FUNCTION TFWAconCodiceWPPPresente : BOOL // Valuta se esiste una WA in lavorazione con il codice del pacco sul ribaltino, se esiste ritorna true, altrimenti false
VAR_INPUT
	WorkArea : POINTER TO ARRAY [1..MAXAREA] OF TFMachinePalletizer_WorkArea;
	WorkAreaState : POINTER TO ARRAY [1..MAXAREA] OF TFMachinePalletizer_WorkAreaState;
	WorkPickPointState : POINTER TO ARRAY [1..MAXPICKPOINT] OF TFMachinePalletizer_WorkPickPointState;
	ppick : INT;
END_VAR
VAR
	wa : INT;
END_VAR

// Valuta se esiste una WA in lavorazione con il codice del pacco sul ribaltino, se esiste ritorna true, altrimenti false
TFWAconCodiceWPPPresente := FALSE;

(* Per tutte le WorkArea Attive e in Lavorazione *)
FOR wa:=1 TO MAXAREA DO
		IF WorkArea^[wa].Enable = 1 THEN
		(* Verifico se è in lavorazione *)
			IF WorkAreaState^[wa].State = WORKAREA_STATE_OCCUPIED_WORKING AND WorkArea^[wa].Typology = TYPOLOGY_PALLET THEN
				(* Verifico se il codice della WA è uguale al codice sul ribaltino *)
				IF WorkAreaState^[wa].Code = WorkPickPointState^[ppick].Code THEN
					TFWAconCodiceWPPPresente := TRUE;
					RETURN;
				END_IF
			END_IF
		END_IF
END_FOR

END_FUNCTION

(* stored: Version 1.1.0.1, ProductVersion 3.1.4024.11
   POU TFWAconCodiceWPPPresente: Id {44eb7b2a-2d69-435e-9f70-759be00d73fa}, SpecialFunc None *)
